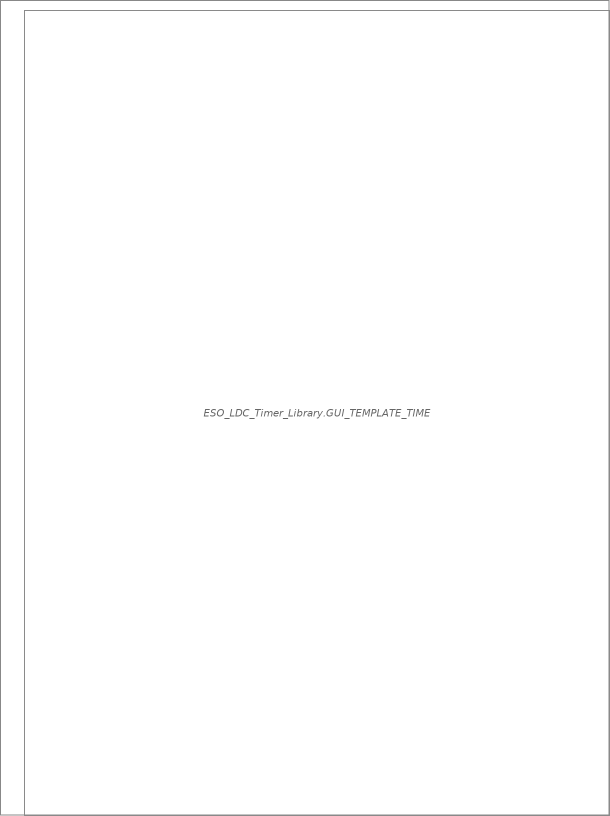
VISUALIZATION GUI_TIMER  // 610x816
    Frame (24,10 586x806)
        shows ESO_LDC_Timer_Library.GUI_TEMPLATE_TIME(m_Instance := MAIN.fbTimer)
END_VISUALIZATION

(* stored: Version 1.1.0.1, ProductVersion 3.1.4024.9
   Visu GUI_TIMER: Id {8f57a1bc-2cb2-4396-b7be-20ce6f4ecd8e} *)
